# EPICS StreamDevice protocol: streamSim/protocols/streamsim.proto
# example stream protocol file

Terminator = CR LF;
ReplyTimeout = 10000; # 10 sec is very long, for keyboard input
ReadTimeout = 1000;   # also long for keyboard input

li {
    out "%(NAME)s?";
    in "%d";
}
